FUNCTION_BLOCK Door (* Composite Function Block Type *)
  (* Standard: 61499-2 *)
  (* Version 0.0, 6/3/2016, Andrei, nxtControl GmbH, template *)
  PACKAGE Main;
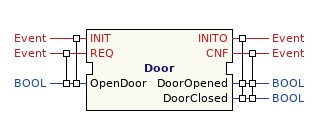
  EVENT_INPUT
    INIT WITH OpenDoor; (* Initialization Request *)
    REQ WITH OpenDoor; (* Normal Execution Request *)
  END_EVENT
  EVENT_OUTPUT
    INITO WITH DoorOpened, DoorClosed; (* Initialization Confirm *)
    CNF WITH DoorOpened, DoorClosed; (* Execution Confirmation *)
  END_EVENT
  VAR_INPUT
    OpenDoor : BOOL; (* Input event qualifier *)
  END_VAR
  VAR_OUTPUT
    DoorOpened : BOOL;
    DoorClosed : BOOL;
  END_VAR
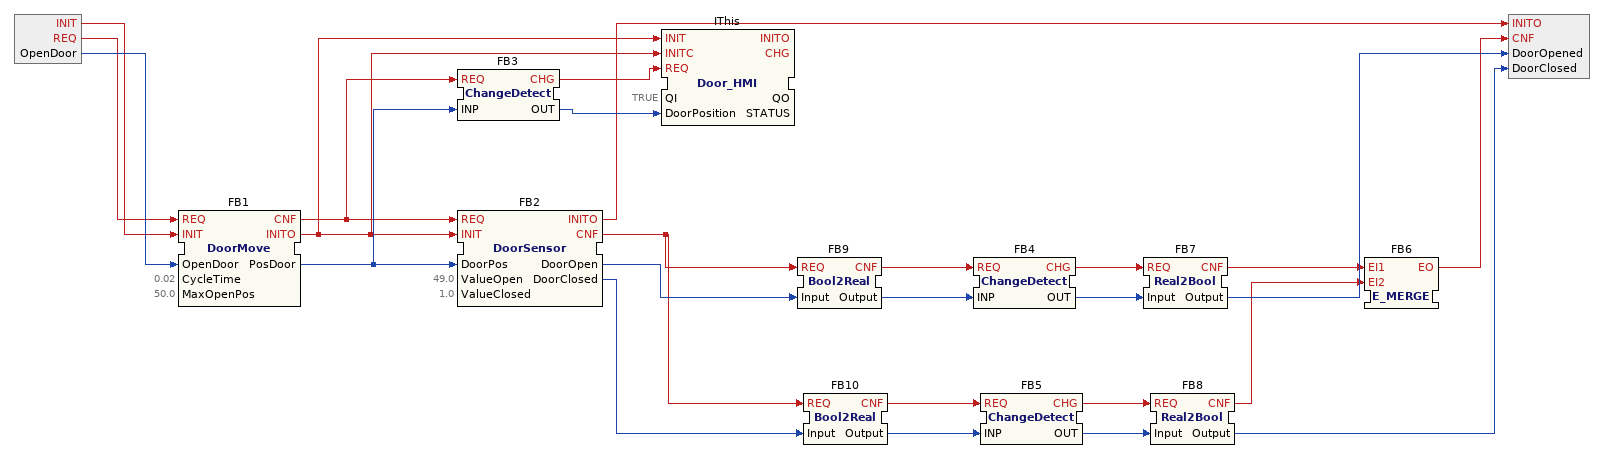
  FBS
    FB2 : DoorSensor(ValueOpen := 49.0, ValueClosed := 1.0);
    FB3 : ChangeDetect;
    FB1 : DoorMove(CycleTime := 0.02, MaxOpenPos := 50.0);
    IThis : Door_HMI(QI := TRUE);
    FB4 : ChangeDetect;
    FB5 : ChangeDetect;
    FB6 : E_MERGE;
    FB7 : Real2Bool;
    FB8 : Real2Bool;
    FB9 : Bool2Real;
    FB10 : Bool2Real;
  END_FBS
  EVENT_CONNECTIONS
    FB1.CNF TO FB2.REQ;
    FB1.INITO TO FB2.INIT;
    FB2.INITO TO INITO;
    REQ TO FB1.REQ;
    INIT TO FB1.INIT;
    FB1.INITO TO IThis.INIT;
    FB3.CHG TO IThis.REQ;
    FB1.CNF TO FB3.REQ;
    FB1.INITO TO IThis.INITC;
    FB2.CNF TO FB9.REQ;
    FB2.CNF TO FB10.REQ;
    FB6.EO TO CNF;
    FB4.CHG TO FB7.REQ;
    FB5.CHG TO FB8.REQ;
    FB7.CNF TO FB6.EI1;
    FB8.CNF TO FB6.EI2;
    FB9.CNF TO FB4.REQ;
    FB10.CNF TO FB5.REQ;
  END_CONNECTIONS
  DATA_CONNECTIONS
    OpenDoor TO FB1.OpenDoor;
    FB1.PosDoor TO FB2.DoorPos;
    FB3.OUT TO IThis.DoorPosition;
    FB1.PosDoor TO FB3.INP;
    FB2.DoorOpen TO FB9.Input;
    FB2.DoorClosed TO FB10.Input;
    FB5.OUT TO FB8.Input;
    FB4.OUT TO FB7.Input;
    FB7.Output TO DoorOpened;
    FB8.Output TO DoorClosed;
    FB9.Output TO FB4.INP;
    FB10.Output TO FB5.INP;
  END_CONNECTIONS
END_FUNCTION_BLOCK
